(* Visualisation Calibrations/ONE_FUEL_CALIBRATION
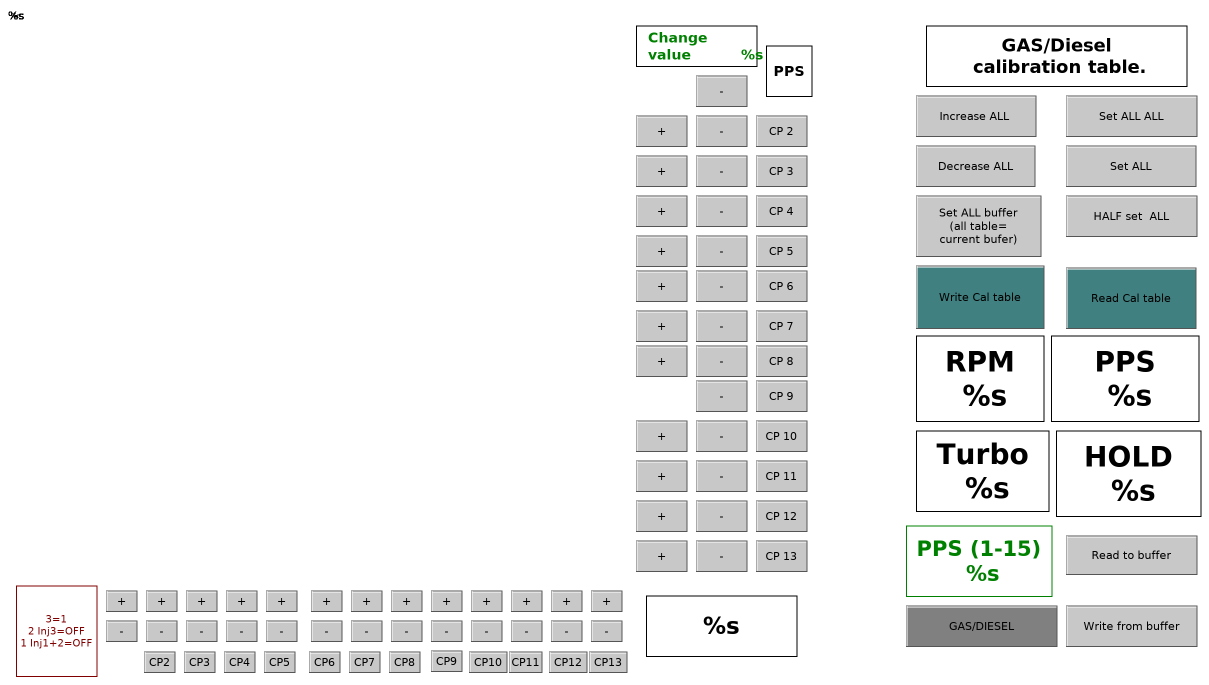
rectangle at (0,0)-(0,0): text "%s"; shows p.RPM_table[INDEX]; editable
rectangle at (0,0)-(0,0): text "%s"; shows p.Turbo_table[1]; editable
rectangle at (0,0)-(0,0): text "%s"; shows p.Turbo_table[2]; editable
rectangle at (0,0)-(0,0): text "%s"; shows p.Turbo_table[3]; editable
rectangle at (0,0)-(0,0): text "%s"; shows p.Turbo_table[4]; editable
rectangle at (0,0)-(0,0): text "%s"; shows p.Turbo_table[5]; editable
rectangle at (0,0)-(0,0): text "%s"; shows p.Turbo_table[6]; editable
rectangle at (0,0)-(0,0): text "%s"; shows p.Turbo_table[7]; editable
rectangle at (0,0)-(0,0): text "%s"; shows p.Turbo_table[8]; editable
rectangle at (0,0)-(0,0): text "%s"; shows p.Turbo_table[9]; editable
rectangle at (0,0)-(0,0): text "%s"; shows p.Turbo_table[10]; editable
rectangle at (0,0)-(0,0): text "%s"; shows p.Turbo_table[11]; editable
rectangle at (0,0)-(0,0): text "%s"; shows p.Turbo_table[12]; editable
rectangle at (0,0)-(0,0): text "%s"; shows p.Turbo_table[13]; editable
rounded rectangle at (890,510)-(1036,581): text "PPS (1-15) / %s"; shows DFPRS_Change_Cal_Table.PPS_number; editable
button at (900,80)-(1020,121): text "Increase ALL"; taps DFPRS_Change_Cal_Table.ALL_plus
button at (900,130)-(1019,171): text "Decrease ALL"; taps DFPRS_Change_Cal_Table.ALL_minus
button at (1050,252)-(1180,313): text "Read Cal table"; taps DFPRS_Change_Cal_Table.Read_cal
button at (900,250)-(1028,313): text "Write Cal table"; taps DFPRS_Change_Cal_Table.Write_cal
button at (1050,130)-(1180,171): text "Set ALL"; taps DFPRS_Change_Cal_Table.Set_ALL
button at (1050,180)-(1181,221): text "HALF set  ALL"; taps DFPRS_Change_Cal_Table.HALF_set_ALL
button at (680,60)-(731,91): text "-"; taps DFPRS_Change_Cal_Table.RPM_Flag_minus_1
button at (620,100)-(671,131): text "+"; taps DFPRS_Change_Cal_Table.RPM_Flag_plus_2
button at (680,100)-(731,131): text "-"; taps DFPRS_Change_Cal_Table.RPM_Flag_minus_2
button at (740,100)-(791,131): text "CP 2"; taps DFPRS_Change_Cal_Table.RPM_Flag_CP_2
button at (620,140)-(671,171): text "+"; taps DFPRS_Change_Cal_Table.RPM_Flag_plus_3
button at (680,140)-(731,171): text "-"; taps DFPRS_Change_Cal_Table.RPM_Flag_minus_3
button at (740,140)-(791,171): text "CP 3"; taps DFPRS_Change_Cal_Table.RPM_Flag_CP_3
button at (620,180)-(671,211): text "+"; taps DFPRS_Change_Cal_Table.RPM_Flag_plus_4
button at (680,180)-(731,211): text "-"; taps DFPRS_Change_Cal_Table.RPM_Flag_minus_4
button at (740,180)-(791,211): text "CP 4"; taps DFPRS_Change_Cal_Table.RPM_Flag_CP_4
button at (620,220)-(671,251): text "+"; taps DFPRS_Change_Cal_Table.RPM_Flag_plus_5
button at (680,220)-(731,251): text "-"; taps DFPRS_Change_Cal_Table.RPM_Flag_minus_5
button at (740,220)-(791,251): text "CP 5"; taps DFPRS_Change_Cal_Table.RPM_Flag_CP_5
button at (620,255)-(671,286): text "+"; taps DFPRS_Change_Cal_Table.RPM_Flag_plus_6
button at (680,255)-(731,286): text "-"; taps DFPRS_Change_Cal_Table.RPM_Flag_minus_6
button at (740,255)-(791,286): text "CP 6"; taps DFPRS_Change_Cal_Table.RPM_Flag_CP_6
button at (620,295)-(671,326): text "+"; taps DFPRS_Change_Cal_Table.RPM_Flag_plus_7
button at (680,295)-(731,326): text "-"; taps DFPRS_Change_Cal_Table.RPM_Flag_minus_7
button at (740,295)-(791,326): text "CP 7"; taps DFPRS_Change_Cal_Table.RPM_Flag_CP_7
button at (620,330)-(671,361): text "+"; taps DFPRS_Change_Cal_Table.RPM_Flag_plus_8
button at (680,330)-(731,361): text "-"; taps DFPRS_Change_Cal_Table.RPM_Flag_minus_8
button at (740,330)-(791,361): text "CP 8"; taps DFPRS_Change_Cal_Table.RPM_Flag_CP_8
button at (90,575)-(121,596): text "+"; taps DFPRS_Change_Cal_Table.Turbo_Flag_plus_1
button at (90,605)-(121,626): text "-"; taps DFPRS_Change_Cal_Table.Turbo_Flag_minus_1
button at (130,575)-(161,596): text "+"; taps DFPRS_Change_Cal_Table.Turbo_Flag_plus_2
button at (130,605)-(161,626): text "-"; taps DFPRS_Change_Cal_Table.Turbo_Flag_minus_2
button at (128,636)-(159,657): text "CP2"; taps DFPRS_Change_Cal_Table.Turbo_Flag_CP_2
button at (170,575)-(201,596): text "+"; taps DFPRS_Change_Cal_Table.Turbo_Flag_plus_3
button at (170,605)-(201,626): text "-"; taps DFPRS_Change_Cal_Table.Turbo_Flag_minus_3
button at (168,636)-(199,657): text "CP3"; taps DFPRS_Change_Cal_Table.Turbo_Flag_CP_3
button at (210,575)-(241,596): text "+"; taps DFPRS_Change_Cal_Table.Turbo_Flag_plus_4
button at (210,605)-(241,626): text "-"; taps DFPRS_Change_Cal_Table.Turbo_Flag_minus_4
button at (208,636)-(239,657): text "CP4"; taps DFPRS_Change_Cal_Table.Turbo_Flag_CP_4
button at (250,575)-(281,596): text "+"; taps DFPRS_Change_Cal_Table.Turbo_Flag_plus_5
button at (250,605)-(281,626): text "-"; taps DFPRS_Change_Cal_Table.Turbo_Flag_minus_5
button at (248,636)-(279,657): text "CP5"; taps DFPRS_Change_Cal_Table.Turbo_Flag_CP_5
button at (295,575)-(326,596): text "+"; taps DFPRS_Change_Cal_Table.Turbo_Flag_plus_6
button at (295,605)-(326,626): text "-"; taps DFPRS_Change_Cal_Table.Turbo_Flag_minus_6
button at (293,636)-(324,657): text "CP6"; taps DFPRS_Change_Cal_Table.Turbo_Flag_CP_6
button at (335,575)-(366,596): text "+"; taps DFPRS_Change_Cal_Table.Turbo_Flag_plus_7
button at (335,605)-(366,626): text "-"; taps DFPRS_Change_Cal_Table.Turbo_Flag_minus_7
button at (333,636)-(364,657): text "CP7"; taps DFPRS_Change_Cal_Table.Turbo_Flag_CP_7
button at (375,575)-(406,596): text "+"; taps DFPRS_Change_Cal_Table.Turbo_Flag_plus_8
button at (375,605)-(406,626): text "-"; taps DFPRS_Change_Cal_Table.Turbo_Flag_minus_8
button at (373,636)-(404,657): text "CP8"; taps DFPRS_Change_Cal_Table.Turbo_Flag_CP_8
rounded rectangle at (620,10)-(741,51): text "Change / value          %s"; shows DFPRS_Change_Cal_Table.Change_volume; editable 0..
rounded rectangle at (1035,320)-(1183,406): text "PPS / %s"; shows .PPS1
rounded rectangle at (1040,415)-(1185,501): text "HOLD / %s"; shows .HOLD_time
rounded rectangle at (910,10)-(1171,71): text "GAS/Diesel / calibration table."
button at (1050,520)-(1181,559): text "Read to buffer"; taps DFPRS_Change_Cal_Table.red_cal2
button at (1050,590)-(1181,631): text "Write from buffer"; taps DFPRS_Change_Cal_Table.Write_cal2
rounded rectangle at (900,320)-(1028,406): text "RPM / %s"; shows .RPM
rounded rectangle at (900,415)-(1033,496): text "Turbo / %s"; shows .Turbo_pressure
rounded rectangle at (750,30)-(796,81): text "PPS"
button at (680,365)-(731,396): text "-"; taps DFPRS_Change_Cal_Table.RPM_Flag_minus_9
button at (620,405)-(671,436): text "+"; taps DFPRS_Change_Cal_Table.RPM_Flag_plus_10
button at (680,405)-(731,436): text "-"; taps DFPRS_Change_Cal_Table.RPM_Flag_minus_10
button at (740,405)-(791,436): text "CP 10"; taps DFPRS_Change_Cal_Table.RPM_Flag_CP_10
button at (620,445)-(671,476): text "+"; taps DFPRS_Change_Cal_Table.RPM_Flag_plus_11
button at (680,445)-(731,476): text "-"; taps DFPRS_Change_Cal_Table.RPM_Flag_minus_11
button at (740,445)-(791,476): text "CP 11"; taps DFPRS_Change_Cal_Table.RPM_Flag_CP_11
button at (620,485)-(671,516): text "+"; taps DFPRS_Change_Cal_Table.RPM_Flag_plus_12
button at (680,485)-(731,516): text "-"; taps DFPRS_Change_Cal_Table.RPM_Flag_minus_12
button at (740,485)-(791,516): text "CP 12"; taps DFPRS_Change_Cal_Table.RPM_Flag_CP_12
button at (620,525)-(671,556): text "+"; taps DFPRS_Change_Cal_Table.RPM_Flag_plus_13
button at (680,525)-(731,556): text "-"; taps DFPRS_Change_Cal_Table.RPM_Flag_minus_13
button at (740,525)-(791,556): text "CP 13"; taps DFPRS_Change_Cal_Table.RPM_Flag_CP_13
button at (740,365)-(791,396): text "CP 9"; taps DFPRS_Change_Cal_Table.RPM_Flag_CP_9
button at (415,575)-(446,596): text "+"; taps DFPRS_Change_Cal_Table.Turbo_Flag_plus_9
button at (415,605)-(446,626): text "-"; taps DFPRS_Change_Cal_Table.Turbo_Flag_minus_9
button at (455,575)-(486,596): text "+"; taps DFPRS_Change_Cal_Table.Turbo_Flag_plus_10
button at (455,605)-(486,626): text "-"; taps DFPRS_Change_Cal_Table.Turbo_Flag_minus_10
button at (453,636)-(491,657): text "CP10"; taps DFPRS_Change_Cal_Table.Turbo_Flag_CP_10
button at (495,575)-(526,596): text "+"; taps DFPRS_Change_Cal_Table.Turbo_Flag_plus_11
button at (495,605)-(526,626): text "-"; taps DFPRS_Change_Cal_Table.Turbo_Flag_minus_11
button at (493,636)-(526,657): text "CP11"; taps DFPRS_Change_Cal_Table.Turbo_Flag_CP_11
button at (535,575)-(566,596): text "+"; taps DFPRS_Change_Cal_Table.Turbo_Flag_plus_12
button at (535,605)-(566,626): text "-"; taps DFPRS_Change_Cal_Table.Turbo_Flag_minus_12
button at (533,636)-(571,657): text "CP12"; taps DFPRS_Change_Cal_Table.Turbo_Flag_CP_12
button at (575,575)-(606,596): text "+"; taps DFPRS_Change_Cal_Table.Turbo_Flag_plus_13
button at (575,605)-(606,626): text "-"; taps DFPRS_Change_Cal_Table.Turbo_Flag_minus_13
button at (573,636)-(611,657): text "CP13"; taps DFPRS_Change_Cal_Table.Turbo_Flag_CP_13
button at (415,635)-(446,656): text "CP9"; taps DFPRS_Change_Cal_Table.Turbo_Flag_CP_9
button at (1050,80)-(1181,121): text "Set ALL ALL"; taps DFPRS_Change_Cal_Table.Set_ALL_ALL
button at (900,180)-(1025,241): text "Set ALL buffer / (all table= / current bufer)"; taps DFPRS_Change_Cal_Table.Set_ALL_ALL
rectangle at (0,570)-(81,661): text "3=1 / 2 Inj3=OFF / 1 Inj1+2=OFF"
rectangle at (0,0)-(0,0): text "%s"; shows p.PPS_table[INDEX]; editable
button at (890,590)-(1041,631): text "GAS/DIESEL"; toggles DFPRS_Change_Cal_Table.Flag_cal_table_gas
rounded rectangle at (630,580)-(781,641): text "%s"; shows DFPRS_Change_Cal_Table.Fuel_type
*)

(* Visualisation PLC_VISU
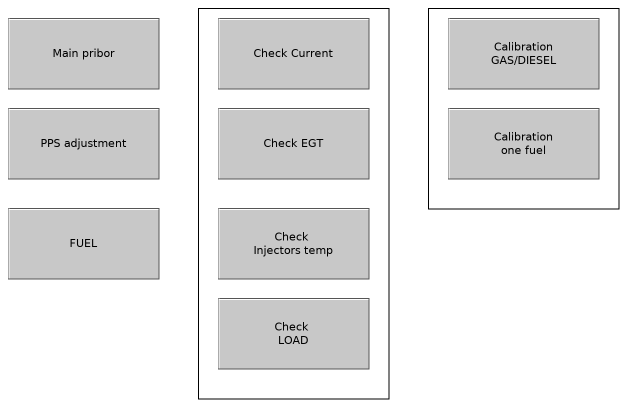
button at (40,30)-(191,101): text "Main pribor"; opens MAIN_PRIBOR
button at (250,30)-(401,101): text "Check Current"; opens CHECK_CURRENT
button at (250,120)-(401,191): text "Check EGT"; opens CHECK_EGT
button at (250,220)-(401,291): text "Check / Injectors temp"; opens CHECK_INJ_TEMP
button at (480,30)-(631,101): text "Calibration / GAS/DIESEL"; opens CALIBRATION_GAS_DIESEL
button at (480,120)-(631,191): text "Calibration / one fuel"; opens ONE_FUEL_CALIBRATION
button at (40,120)-(191,191): text "PPS adjustment"; opens PPS_PWM_adjustment
button at (40,220)-(191,291): text "FUEL"; opens FUEL
button at (250,310)-(401,381): text "Check / LOAD"; opens CHECK_Load
2 more shapes without text or variables
*)

(* Visualisation PPS_PWM_adjustment
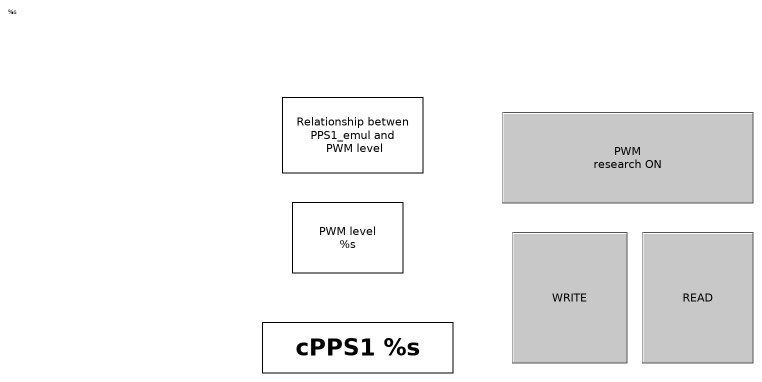
button at (490,100)-(741,191): text "PWM / research ON"; toggles .Flag_PWM_researh
button at (500,220)-(615,351): text "WRITE"; taps DFPRS_Change_Cal_Table.Write_cal
button at (630,220)-(741,351): text "READ"; taps DFPRS_Change_Cal_Table.Read_cal
rounded rectangle at (270,85)-(411,161): text "Relationship betwen / PPS1_emul and / PWM level"
rounded rectangle at (280,190)-(391,261): text "PWM level / %s"; shows Act_control.j; editable
rectangle at (0,0)-(0,0): text "%s"; shows p.PPS1_emul_PWM[INDEX]; editable
rounded rectangle at (250,310)-(441,361): text "cPPS1 %s"; shows .cPPS1_emul
1 elements of other kinds (tables, trends, ...) not read
*)

(* Visualisation SETUP
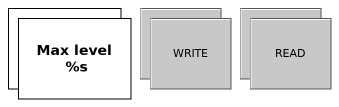
rounded rectangle at (1018,710)-(1131,791): text "Max level / %s"; shows .p.EGT_max; editable
button at (1250,710)-(1331,781): text "READ"; taps DFPRS_Change_Cal_Table.Read_cal
button at (1150,710)-(1231,781): text "WRITE"; taps DFPRS_Change_Cal_Table.Write_cal
rounded rectangle at (1028,720)-(1141,801): text "Max level / %s"; shows .p.EGT_max; editable
button at (1260,720)-(1341,791): text "READ"; taps DFPRS_Change_Cal_Table.Read_cal
button at (1160,720)-(1241,791): text "WRITE"; taps DFPRS_Change_Cal_Table.Write_cal
*)
